// TIA Portal project "CommRS485" (V17)

(* hardware
DEVICE "S7-1200 station_1"  S7-1200 Station
   slot 0: "Rack_0"  S7-1200 Rack  Rack  V1.0
   slot 1: "PLC_1"  CPU 1211C DC/DC/Rly  6ES7 211-1HE40-0XB0  V4.5
   slot 101: "CM 1241 (RS422/485)_1"  6ES7 241-1CH32-0XB0  V2.2
DEVICE "S7-1200 station_2"  S7-1200 Station
   slot 0: "Rack_0"  S7-1200 Rack  Rack  V1.0
   slot 1: "PLC_2"  CPU 1215C AC/DC/Rly  6ES7 215-1BG31-0XB0  V3.0
   slot 3: "AQ 1x12BIT_1"  AQ1 signal board  6ES7 232-4HA30-0XB0  V1.0
   slot 101: "CM 1241 (RS485)_1"  CM 1241 (RS485)  6ES7 241-1CH30-0XB0  V1.0
DEVICE "HMI_1"  KTP400 Comfort
   slot 0: "HMI_1"  KTP400 Comfort  6AV2 124-2DC01-0AX0  17.0.0.0
   slot 1: "HMI_RT_1"  KTP400 Comfort  6AV2 124-2DC01-0AX0  17.0.0.0
   slot 5: "HMI_1.IE_CP_1"  PROFINET Interface  17.0.0.0
      slot 1: "PROFINET Interface_1"  PROFINET Interface
         slot 1: "Port_1"  Port
   slot 7: "HMI_1.MPI/DP_CP_1"  MPI/DP Interface  17.0.0.0
*)

// ===== PLC "PLC_1"  CPU 1211C DC/DC/Rly =====

VAR_GLOBAL   // PLC tag table "Default tag table"
   "FirstScan" AT %M1.0 : Bool;
   "DiagStatusUpdate" AT %M1.1 : Bool;
   "AlwaysTRUE" AT %M1.2 : Bool;
   "Clock_Byte" AT %MB1 : Byte;
   "Clock_2Hz" AT %M1.3 : Bool;
   "Clock_1.25Hz" AT %M1.4 : Bool;
   "Clock_1Hz" AT %M1.5 : Bool;
   "Clock_0.625Hz" AT %M1.6 : Bool;
   "Clock_0.5Hz" AT %M1.7 : Bool;
   "MODE_MASTER" AT %M2.0 : Bool;
   "scanOne" AT %M2.1 : Bool;
   "Tag_1" AT %M4.0 : Bool;
   "Mode_SLAVE" AT %M4.1 : Bool;
   "Tag_2" AT %M2.2 : Bool;
   "Tag_3" AT %M4.2 : Bool;
   "Clock_Byte(1)" AT %MB0 : Byte;
   "Clock_10Hz(1)" AT %M0.0 : Bool;
   "Clock_5Hz(1)" AT %M0.1 : Bool;
   "Clock_2.5Hz(1)" AT %M0.2 : Bool;
   "Clock_2Hz(1)" AT %M0.3 : Bool;
   "Clock_1.25Hz(1)" AT %M0.4 : Bool;
   "Clock_1Hz(1)" AT %M0.5 : Bool;
   "Clock_0.625Hz(1)" AT %M0.6 : Bool;
   "Clock_0.5Hz(1)" AT %M0.7 : Bool;
   "Read_Input" AT %M2.3 : Bool;
   "Write_OutPut" AT %M2.4 : Bool;
   "LectureBusy" AT %M2.5 : Bool;
   "EcritureBusy" AT %M2.6 : Bool;
   "DoneEcriture" AT %M2.7 : Bool;
   "DoneLecture" AT %M3.0 : Bool;
   "ENTREE_0" AT %I0.0 : Bool;
   "ENTREE_1" AT %I0.1 : Bool;
   "ENTREE_2" AT %I0.2 : Bool;
   "ENTREE_3" AT %I0.3 : Bool;
   "ENTREE_4" AT %I0.4 : Bool;
   "ENTREE_5" AT %I0.5 : Bool;
END_VAR

DATA_BLOCK "MBLOAD_Matser"   // DB1
{ S7_Optimized_Access := 'FALSE' }
VERSION : 0.1
   VAR
      Baud : UDInt := 9600;
      PARITY : UInt;
      DONE : Bool;
      ERROR : Bool;
      STATUS : Word;
   END_VAR
BEGIN
END_DATA_BLOCK

DATA_BLOCK "MBCONFIG_Master"   // DB2
{ S7_Optimized_Access := 'FALSE' }
VERSION : 0.1
   VAR
      REQ : Bool;
      AGAIN : Bool;
      MB_ADDR : UInt := 1;   // DEFAULT ADRESS : 1
      MODE : USInt;   // READ ONLY : 0
      DATA_ADDR : UDInt := 10001;   // STARTING ADRESS : 40001
      DATA_LEN : UInt := 10;   // DATA LENGTH : 10 WORDS
      DONE : Bool;
      ERROR : Bool;
      BUSY : Bool;
      Register_Input : Array[0..9] of Bool;
      STATUS : Word;
   END_VAR
BEGIN
END_DATA_BLOCK

DATA_BLOCK "DATA_BUFF_Master"   // DB3
{ S7_Optimized_Access := 'FALSE' }
VERSION : 0.1
   VAR
      REGISTERS : Array[0..9] of Bool;
   END_VAR
BEGIN
END_DATA_BLOCK

DATA_BLOCK "DATA_BUFF_INPUT"   // DB10
{ S7_Optimized_Access := 'FALSE' }
VERSION : 0.1
   VAR
      REGISTERS : Array[0..9] of Bool;
   END_VAR
BEGIN
END_DATA_BLOCK

DATA_BLOCK "DATA_BUFF_OUTPUT"   // DB11
{ S7_Optimized_Access := 'FALSE' }
VERSION : 0.1
   VAR
      REGISTERS : Array[0..9] of Bool;
   END_VAR
BEGIN
END_DATA_BLOCK

// folder: System blocks/Program resources

DATA_BLOCK "IEC_Timer_0_DB"   // DB6
{ S7_Optimized_Access := 'TRUE' }
AUTHOR : Simatic
FAMILY : IEC
NAME : IEC_TMR
VERSION : 1.0
// stored: InstanceOfName IEC_TIMER
"IEC_TIMER"
BEGIN
END_DATA_BLOCK

DATA_BLOCK "IEC_Timer_0_DB_2"   // DB8
{ S7_Optimized_Access := 'TRUE' }
AUTHOR : Simatic
FAMILY : IEC
NAME : IEC_TMR
VERSION : 1.0
// stored: InstanceOfName IEC_TIMER
"IEC_TIMER"
BEGIN
END_DATA_BLOCK

// folder: (top level)

FUNCTION "REQ_Master_To_Slave" : Void   // FC1, LAD
{ S7_Optimized_Access := 'TRUE' }
VERSION : 0.1
   VAR_TEMP
      done : Bool;
   END_VAR
BEGIN

REGION Network 2: Lecture des entrées
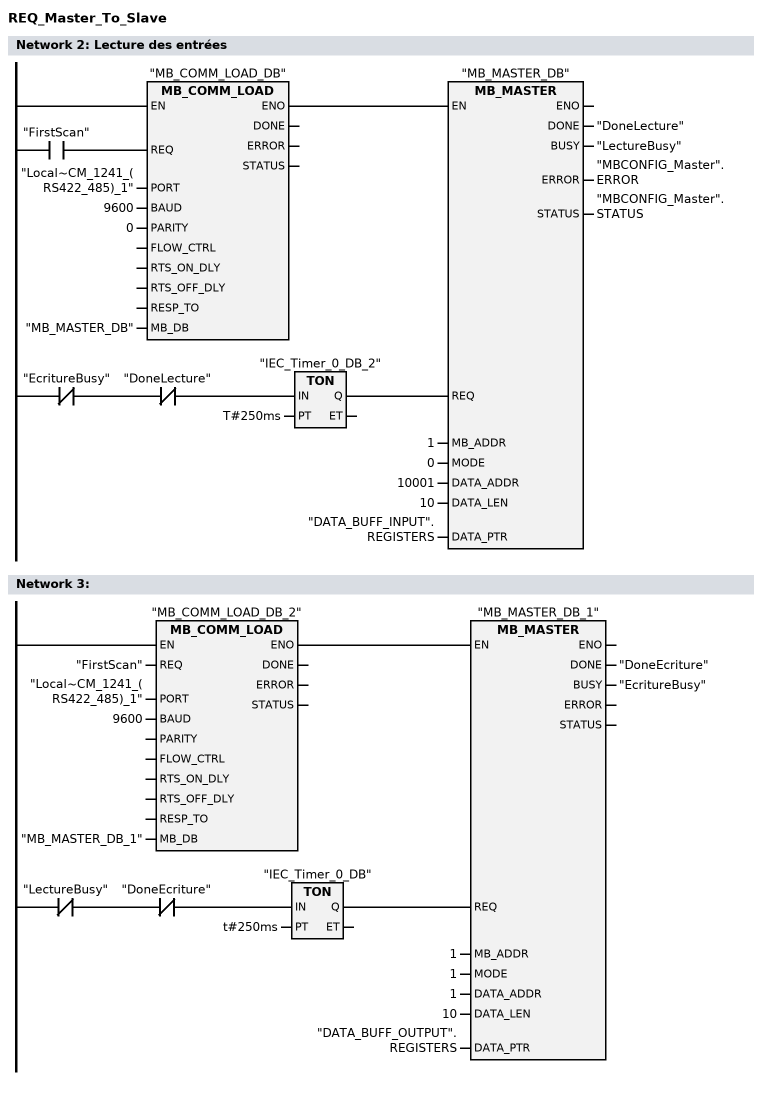
   // ENO of a box is taken as its EN; it also drops when the box reports an error
   "MB_COMM_LOAD_DB"(REQ := "FirstScan",   // MB_COMM_LOAD
                     PORT := "Local~CM_1241_(RS422_485)_1",
                     BAUD := 9600,
                     PARITY := 0,
                     MB_DB := "MB_MASTER_DB");
   "IEC_Timer_0_DB_2".TON(IN := NOT "EcritureBusy" AND NOT "DoneLecture", PT := T#250ms);
   "MB_MASTER_DB"(REQ := "IEC_Timer_0_DB_2".Q,   // MB_MASTER
                  MB_ADDR := 1,
                  MODE := 0,
                  DATA_ADDR := 10001,
                  DATA_LEN := 10,
                  DATA_PTR := "DATA_BUFF_INPUT".REGISTERS,
                  DONE => "DoneLecture",
                  BUSY => "LectureBusy",
                  ERROR => "MBCONFIG_Master".ERROR,
                  STATUS => "MBCONFIG_Master".STATUS);
END_REGION

REGION Network 3
   // ENO of a box is taken as its EN; it also drops when the box reports an error
   "MB_COMM_LOAD_DB_2"(REQ := "FirstScan",   // MB_COMM_LOAD
                       PORT := "Local~CM_1241_(RS422_485)_1",
                       BAUD := 9600,
                       MB_DB := "MB_MASTER_DB_1");
   "IEC_Timer_0_DB".TON(IN := NOT "LectureBusy" AND NOT "DoneEcriture", PT := t#250ms);
   "MB_MASTER_DB_1"(REQ := "IEC_Timer_0_DB".Q,   // MB_MASTER
                    MB_ADDR := 1,
                    MODE := 1,
                    DATA_ADDR := 1,
                    DATA_LEN := 10,
                    DATA_PTR := "DATA_BUFF_OUTPUT".REGISTERS,
                    DONE => "DoneEcriture",
                    BUSY => "EcritureBusy");
END_REGION
END_FUNCTION

FUNCTION "ForcageSortie" : Void   // FC3, LAD
{ S7_Optimized_Access := 'TRUE' }
VERSION : 0.1
BEGIN

REGION Network 1
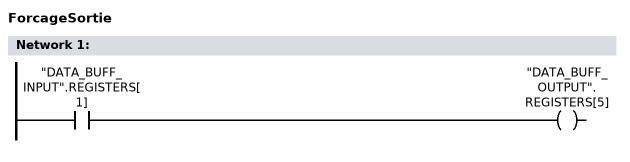
   RUNG wire#powerrail
      Contact( "DATA_BUFF_INPUT".REGISTERS[1] )
      Coil( "DATA_BUFF_OUTPUT".REGISTERS[5] )
   END_RUNG
   // the same network as SCL:
   "DATA_BUFF_OUTPUT".REGISTERS[5] := "DATA_BUFF_INPUT".REGISTERS[1];
END_REGION
END_FUNCTION

ORGANIZATION_BLOCK "Main"   // OB1, LAD, ProgramCycle
TITLE = "Main Program Sweep (Cycle)"
{ S7_Optimized_Access := 'TRUE' }
VERSION : 0.1
   VAR_INPUT
      Initial_Call : Bool;   // Initial call of this OB
      Remanence : Bool;   // =True, if remanent data are available
   END_VAR
BEGIN

REGION Network 1: Call Request Master To Slave
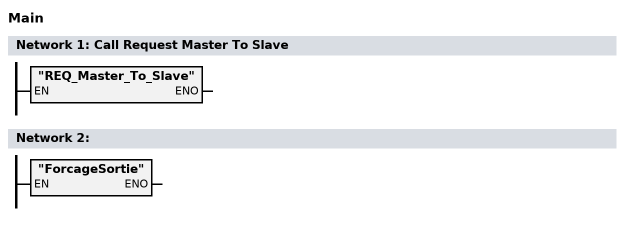
   RUNG wire#powerrail
      "REQ_Master_To_Slave"()
   END_RUNG
   // the same network as SCL:
   "REQ_Master_To_Slave"();
END_REGION

REGION Network 2
   RUNG wire#powerrail
      "ForcageSortie"()
   END_RUNG
   // the same network as SCL:
   "ForcageSortie"();
END_REGION
END_ORGANIZATION_BLOCK

// ===== PLC "PLC_2"  CPU 1215C AC/DC/Rly =====

VAR_GLOBAL   // PLC tag table "Default tag table"
   "System_Byte" AT %MB1 : Byte;
   "FirstScan" AT %M1.0 : Bool;
   "DiagStatusUpdate" AT %M1.1 : Bool;
   "AlwaysTRUE" AT %M1.2 : Bool;
   "AlwaysFALSE" AT %M1.3 : Bool;
   "Clock_Byte" AT %MB0 : Byte;
   "Clock_10Hz" AT %M0.0 : Bool;
   "Clock_5Hz" AT %M0.1 : Bool;
   "Clock_2.5Hz" AT %M0.2 : Bool;
   "Clock_2Hz" AT %M0.3 : Bool;
   "Clock_1.25Hz" AT %M0.4 : Bool;
   "Clock_1Hz" AT %M0.5 : Bool;
   "Clock_0.625Hz" AT %M0.6 : Bool;
   "Clock_0.5Hz" AT %M0.7 : Bool;
END_VAR

DATA_BLOCK "MB_LOAD_SLAVE"   // DB1
{ S7_Optimized_Access := 'FALSE' }
VERSION : 0.1
   VAR
      Baud : UDInt := 9600;
      PARITY : UInt;
      DONE : Bool;
      ERROR : Bool;
      STATUS : Word;
   END_VAR
BEGIN
END_DATA_BLOCK

DATA_BLOCK "MB_CONFIG_SLAVE"   // DB2
{ S7_Optimized_Access := 'FALSE' }
VERSION : 0.1
   VAR
      MB_ADDR : UInt := 1;
   END_VAR
BEGIN
END_DATA_BLOCK

DATA_BLOCK "DATA_BUFF_SLAVE"   // DB3
{ S7_Optimized_Access := 'FALSE' }
VERSION : 0.1
   VAR
      REGISTERS : Array[0..9] of Bool;
   END_VAR
BEGIN
END_DATA_BLOCK

FUNCTION "REQ_SLAVE_FROM_MASTER" : Void   // FC1, LAD
{ S7_Optimized_Access := 'TRUE' }
VERSION : 0.1
BEGIN

REGION Network 1
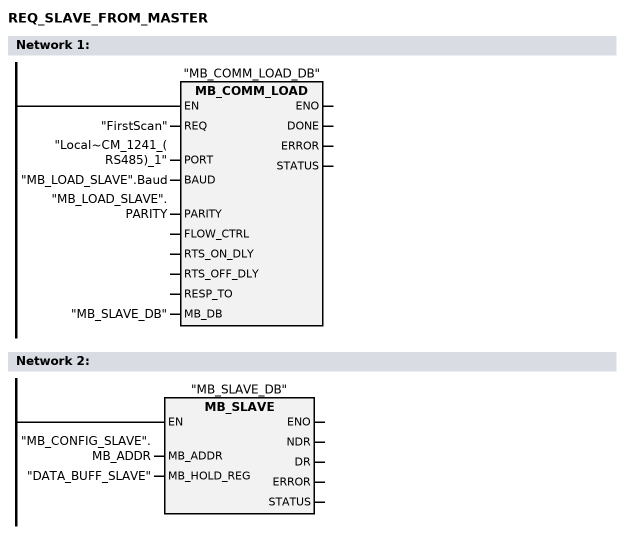
   "MB_COMM_LOAD_DB"(REQ := "FirstScan",   // MB_COMM_LOAD
                     PORT := "Local~CM_1241_(RS485)_1",
                     BAUD := "MB_LOAD_SLAVE".Baud,
                     PARITY := "MB_LOAD_SLAVE".PARITY,
                     MB_DB := "MB_SLAVE_DB");
END_REGION

REGION Network 2
   "MB_SLAVE_DB"(MB_ADDR := "MB_CONFIG_SLAVE".MB_ADDR, MB_HOLD_REG := "DATA_BUFF_SLAVE");   // MB_SLAVE
END_REGION
END_FUNCTION

ORGANIZATION_BLOCK "Main"   // OB1, LAD, ProgramCycle
TITLE = "Main Program Sweep (Cycle)"
{ S7_Optimized_Access := 'TRUE' }
VERSION : 0.1
BEGIN

REGION Network 1
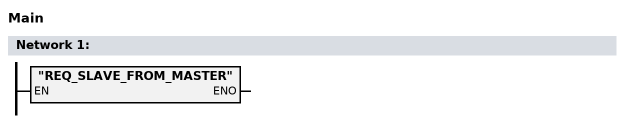
   RUNG wire#powerrail
      "REQ_SLAVE_FROM_MASTER"()
   END_RUNG
   // the same network as SCL:
   "REQ_SLAVE_FROM_MASTER"();
END_REGION
END_ORGANIZATION_BLOCK

(* ===== HMI "HMI_RT_1" =====
system functions are stored by id; their names below are inferred from use

HMI tags "Default tag table"
   "Tag_ScreenNumber" : UInt, internal

Template "Template_1" 480x212
   Button "Exit" at 379,148 size 63x63; TextOff 'Exit'; PictureOff "ExitRuntime_KTP400_Comfort_TR"; PictureOn "ExitRuntime_KTP400_Comfort_TR"
      on Release: StopRuntime(0)
   Button "Template_Button" at 265,148 size 63x63; TextOff 'Text'
   Button "Alarms" at 151,148 size 63x63; TextOff 'Alarms'; PictureOff "AlarmDisplay_KTP400_Comfort_TR"; PictureOn "AlarmDisplay_KTP400_Comfort_TR"
      on Release: function_ef3f5d25("Alarm window_Unacknowledged", -1)
   Button "Start screen" at 37,148 size 63x63; TextOff 'Start screen'; PictureOff "NavigateHome_KTP400_Comfort_TR"; PictureOn "NavigateHome_KTP400_Comfort_TR"
      on Release: ActivateScreen("Screen_1", 0)

screen "Screen_1" 480x212
   Button "Button_1" at 5,163 size 47x48; TextOff 'CmdE'
   Button "Button_2" at 418,3 size 47x48; TextOff 'CmdS'
   Button "Button_3" at 18,27 size 40x65; TextOff 'C2S'
   Button "Button_4" at 221,28 size 40x61; TextOff 'C1S'
   Button "Button_5" at 175,135 size 40x67; TextOff 'C1E'
   Button "Button_6" at 305,131 size 40x71; TextOff 'C2E'
   Button "Button_7" at 417,131 size 40x71; TextOff 'C3E'
   TextField "Text field_1" at 358,45 size 37x20; Text 'CBS'
   TextField "Text field_2" at 363,154 size 37x20; Text 'CBE'
   Group "Group" at 82,126 size 74x76
   Group "Group_1" at 273,20 size 74x76
*)